FUNCTION WORD_TO_SIZE : ST_SIZE
VAR_INPUT
	nValue : WORD;
END_VAR

WORD_TO_SIZE.nValue := nValue;

END_FUNCTION

(* stored: Version 1.1.0.1, ProductVersion 3.1.4024.15
   POU WORD_TO_SIZE: Id {9dff1bdf-2064-485c-9750-00be1ec72651}, SpecialFunc None *)
